% RSLogix 500 project CHIZOM SCADA MAIN.RSS %
PROJECT "UNTITLED"    % processor: MicroLogix 1000 %

PROGRAM FILES
  LAD 2 "MAIN_PROG"  36 rungs
  LAD 3 "USER_FAULT"  1 rungs
  LAD 4 "HSC_INT"  1 rungs
  LAD 5 "STI_INT"  1 rungs
  LAD 6, 7, 8, 9, 10, 11, 12, 13, 14, 15, 16: only END

DATA FILES
  O0 OUTPUT  1 elements
  I1 INPUT  2 elements
  S2 STATUS  33 elements
  B3 BINARY  32 elements
  T4 TIMER  40 elements
  C5 COUNTER  32 elements
  R6 CONTROL  16 elements
  N7 INTEGER  105 elements

LADDER 2 "MAIN_PROG"
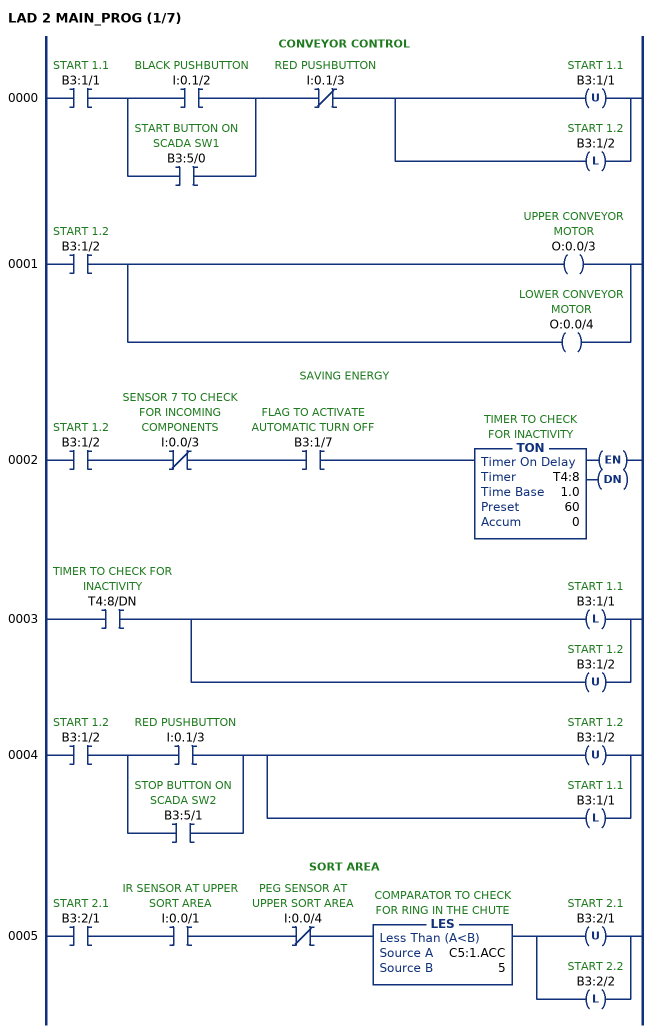
% Rung: 0 %
% TITLE: CONVEYOR CONTROL %
SOR XIC B3:1/1 BST XIC I:0.1/2 NXB XIC B3:5/0 BND XIO I:0.1/3 BST OTU B3:1/1 NXB OTL B3:1/2 BND EOR
%   B3:1/1  "START 1.1" %
%   I:0.1/2  "BLACK PUSHBUTTON" %
%   B3:5/0  SW1  "START BUTTON ON SCADA" %
%   I:0.1/3  "RED PUSHBUTTON" %
%   B3:1/2  "START 1.2" %
% Rung: 1 %
SOR XIC B3:1/2 BST OTE O:0.0/3 NXB OTE O:0.0/4 BND EOR
%   B3:1/2  "START 1.2" %
%   O:0.0/3  "UPPER CONVEYOR MOTOR" %
%   O:0.0/4  "LOWER CONVEYOR MOTOR" %
% Rung: 2 %
% SAVING ENERGY %
SOR XIC B3:1/2 XIO I:0.0/3 XIC B3:1/7 TON T4:8 1.0 60 0 EOR
%   B3:1/2  "START 1.2" %
%   I:0.0/3  "SENSOR 7 TO CHECK FOR INCOMING COMPONENTS" %
%   B3:1/7  "FLAG TO ACTIVATE AUTOMATIC TURN OFF" %
%   T4:8  "TIMER TO CHECK FOR INACTIVITY" %
% Rung: 3 %
SOR XIC T4:8/DN BST OTL B3:1/1 NXB OTU B3:1/2 BND EOR
%   T4:8  "TIMER TO CHECK FOR INACTIVITY" %
%   B3:1/1  "START 1.1" %
%   B3:1/2  "START 1.2" %
% Rung: 4 %
SOR XIC B3:1/2 BST XIC I:0.1/3 NXB XIC B3:5/1 BND BST OTU B3:1/2 NXB OTL B3:1/1 BND EOR
%   B3:1/2  "START 1.2" %
%   I:0.1/3  "RED PUSHBUTTON" %
%   B3:5/1  SW2  "STOP BUTTON ON SCADA" %
%   B3:1/1  "START 1.1" %
% Rung: 5 %
% TITLE: SORT AREA %
SOR XIC B3:2/1 XIC I:0.0/1 XIO I:0.0/4 LES C5:1.ACC 5 BST OTU B3:2/1 NXB OTL B3:2/2 BND EOR
%   B3:2/1  "START 2.1" %
%   I:0.0/1  "IR SENSOR AT UPPER SORT AREA" %
%   I:0.0/4  "PEG SENSOR AT UPPER SORT AREA" %
%   C5:1.ACC  "COMPARATOR TO CHECK FOR RING IN THE CHUTE" %
%   B3:2/2  "START 2.2" %

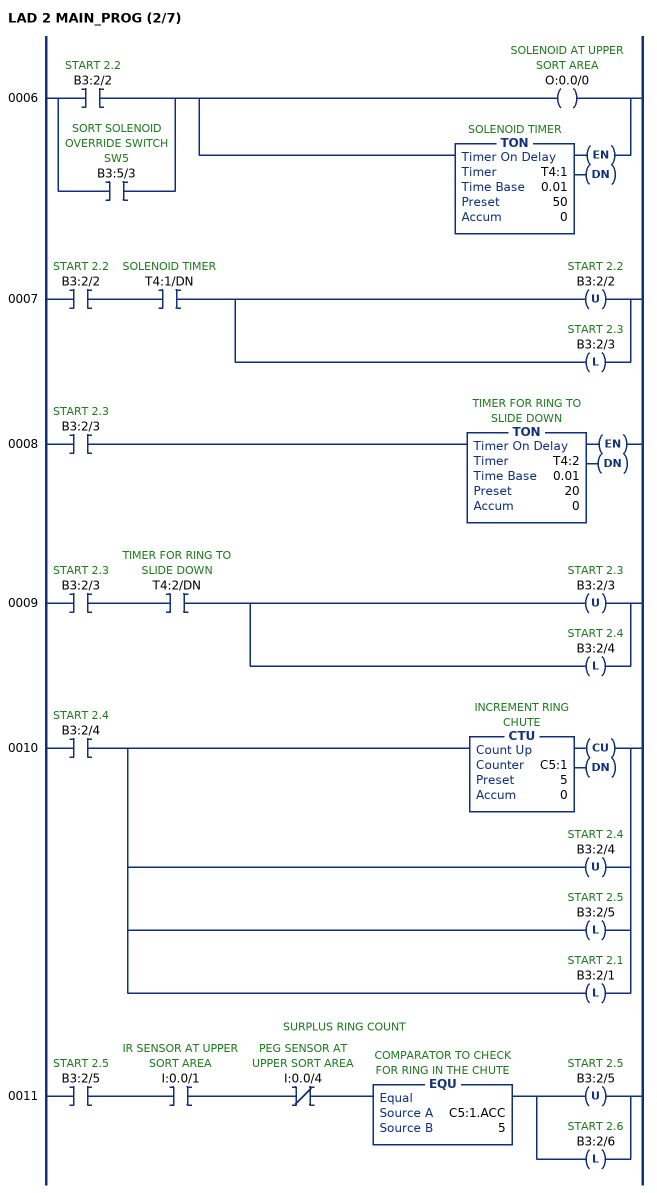
% Rung: 6 %
SOR BST XIC B3:2/2 NXB XIC B3:5/3 BND BST OTE O:0.0/0 NXB TON T4:1 0.01 50 0 BND EOR
%   B3:2/2  "START 2.2" %
%   B3:5/3  SW5  "SORT SOLENOID OVERRIDE SWITCH" %
%   O:0.0/0  "SOLENOID AT UPPER SORT AREA" %
%   T4:1  "SOLENOID TIMER" %
% Rung: 7 %
SOR XIC B3:2/2 XIC T4:1/DN BST OTU B3:2/2 NXB OTL B3:2/3 BND EOR
%   B3:2/2  "START 2.2" %
%   T4:1  "SOLENOID TIMER" %
%   B3:2/3  "START 2.3" %
% Rung: 8 %
SOR XIC B3:2/3 TON T4:2 0.01 20 0 EOR
%   B3:2/3  "START 2.3" %
%   T4:2  "TIMER FOR RING TO SLIDE DOWN" %
% Rung: 9 %
SOR XIC B3:2/3 XIC T4:2/DN BST OTU B3:2/3 NXB OTL B3:2/4 BND EOR
%   B3:2/3  "START 2.3" %
%   T4:2  "TIMER FOR RING TO SLIDE DOWN" %
%   B3:2/4  "START 2.4" %
% Rung: 10 %
SOR XIC B3:2/4 BST CTU C5:1 5 0 NXB BST OTU B3:2/4 NXB BST OTL B3:2/5 NXB OTL B3:2/1 BND BND BND EOR
%   B3:2/4  "START 2.4" %
%   C5:1  "INCREMENT RING CHUTE" %
%   B3:2/5  "START 2.5" %
%   B3:2/1  "START 2.1" %
% Rung: 11 %
% SURPLUS RING COUNT %
SOR XIC B3:2/5 XIC I:0.0/1 XIO I:0.0/4 EQU C5:1.ACC 5 BST OTU B3:2/5 NXB OTL B3:2/6 BND EOR
%   B3:2/5  "START 2.5" %
%   I:0.0/1  "IR SENSOR AT UPPER SORT AREA" %
%   I:0.0/4  "PEG SENSOR AT UPPER SORT AREA" %
%   C5:1.ACC  "COMPARATOR TO CHECK FOR RING IN THE CHUTE" %
%   B3:2/6  "START 2.6" %

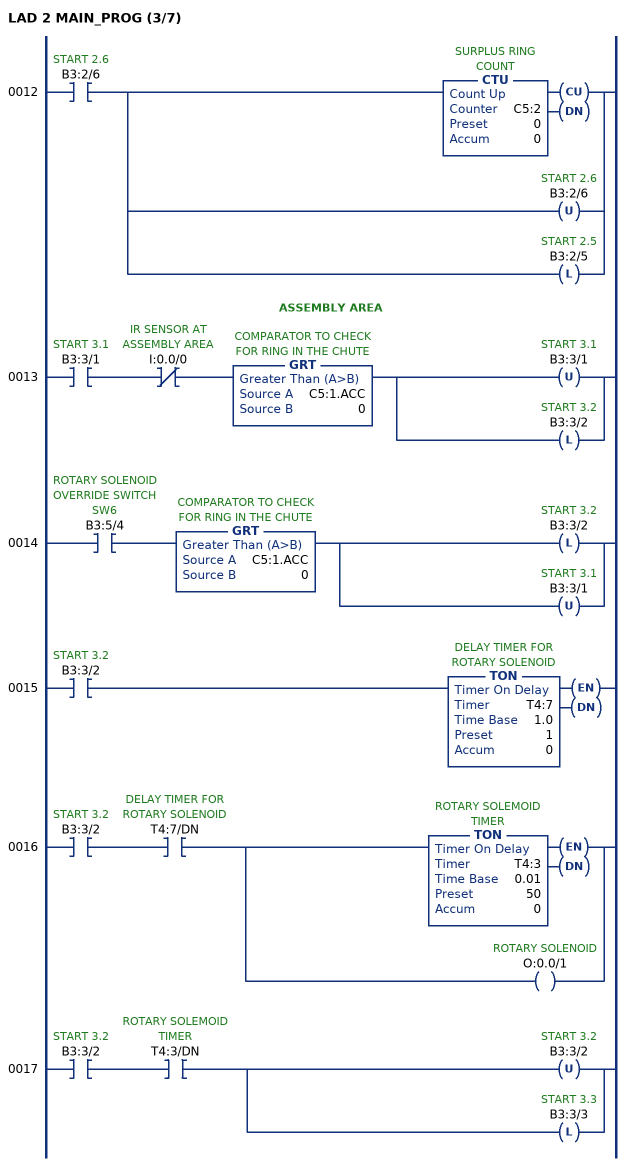
% Rung: 12 %
SOR XIC B3:2/6 BST CTU C5:2 0 0 NXB BST OTU B3:2/6 NXB OTL B3:2/5 BND BND EOR
%   B3:2/6  "START 2.6" %
%   C5:2  "SURPLUS RING COUNT" %
%   B3:2/5  "START 2.5" %
% Rung: 13 %
% TITLE: ASSEMBLY AREA %
SOR XIC B3:3/1 XIO I:0.0/0 GRT C5:1.ACC 0 BST OTU B3:3/1 NXB OTL B3:3/2 BND EOR
%   B3:3/1  "START 3.1" %
%   I:0.0/0  "IR SENSOR AT ASSEMBLY AREA" %
%   C5:1.ACC  "COMPARATOR TO CHECK FOR RING IN THE CHUTE" %
%   B3:3/2  "START 3.2" %
% Rung: 14 %
SOR XIC B3:5/4 GRT C5:1.ACC 0 BST OTL B3:3/2 NXB OTU B3:3/1 BND EOR
%   B3:5/4  SW6  "ROTARY SOLENOID OVERRIDE SWITCH" %
%   C5:1.ACC  "COMPARATOR TO CHECK FOR RING IN THE CHUTE" %
%   B3:3/2  "START 3.2" %
%   B3:3/1  "START 3.1" %
% Rung: 15 %
SOR XIC B3:3/2 TON T4:7 1.0 1 0 EOR
%   B3:3/2  "START 3.2" %
%   T4:7  "DELAY TIMER FOR ROTARY SOLENOID" %
% Rung: 16 %
SOR XIC B3:3/2 XIC T4:7/DN BST TON T4:3 0.01 50 0 NXB OTE O:0.0/1 BND EOR
%   B3:3/2  "START 3.2" %
%   T4:7  "DELAY TIMER FOR ROTARY SOLENOID" %
%   T4:3  "ROTARY SOLEMOID TIMER" %
%   O:0.0/1  "ROTARY SOLENOID" %
% Rung: 17 %
SOR XIC B3:3/2 XIC T4:3/DN BST OTU B3:3/2 NXB OTL B3:3/3 BND EOR
%   B3:3/2  "START 3.2" %
%   T4:3  "ROTARY SOLEMOID TIMER" %
%   B3:3/3  "START 3.3" %

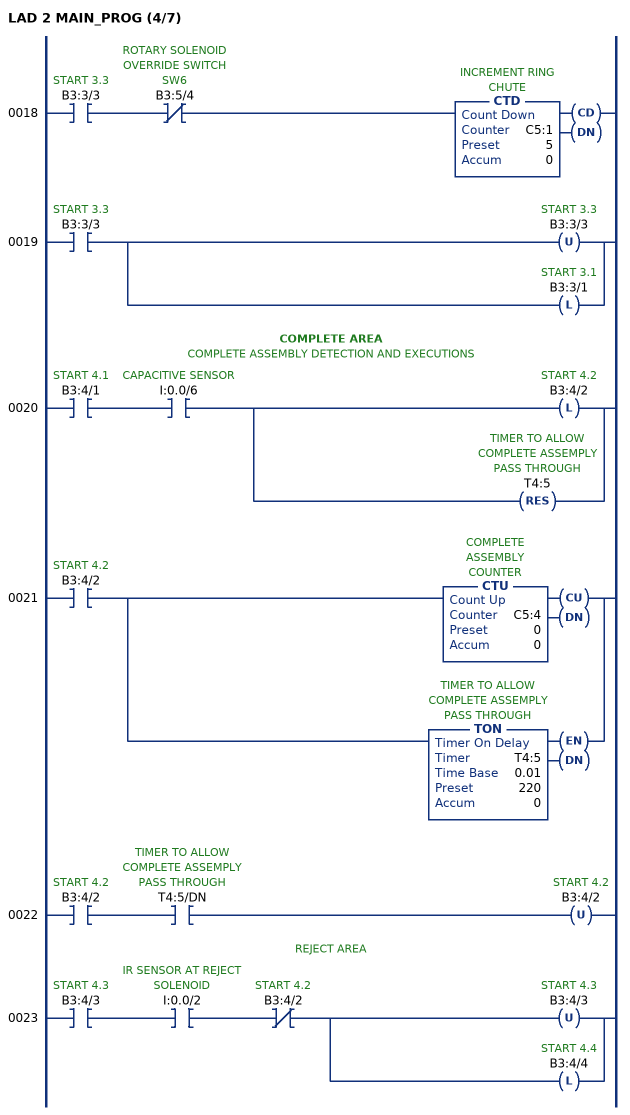
% Rung: 18 %
SOR XIC B3:3/3 XIO B3:5/4 CTD C5:1 5 0 EOR
%   B3:3/3  "START 3.3" %
%   B3:5/4  SW6  "ROTARY SOLENOID OVERRIDE SWITCH" %
%   C5:1  "INCREMENT RING CHUTE" %
% Rung: 19 %
SOR XIC B3:3/3 BST OTU B3:3/3 NXB OTL B3:3/1 BND EOR
%   B3:3/3  "START 3.3" %
%   B3:3/1  "START 3.1" %
% Rung: 20 %
% TITLE: COMPLETE AREA %
% COMPLETE ASSEMBLY DETECTION AND EXECUTIONS %
SOR XIC B3:4/1 XIC I:0.0/6 BST OTL B3:4/2 NXB RES T4:5 BND EOR
%   B3:4/1  "START 4.1" %
%   I:0.0/6  "CAPACITIVE SENSOR" %
%   B3:4/2  "START 4.2" %
%   T4:5  "TIMER TO ALLOW COMPLETE ASSEMPLY PASS THROUGH" %
% Rung: 21 %
SOR XIC B3:4/2 BST CTU C5:4 0 0 NXB TON T4:5 0.01 220 0 BND EOR
%   B3:4/2  "START 4.2" %
%   C5:4  "COMPLETE ASSEMBLY COUNTER" %
%   T4:5  "TIMER TO ALLOW COMPLETE ASSEMPLY PASS THROUGH" %
% Rung: 22 %
SOR XIC B3:4/2 XIC T4:5/DN OTU B3:4/2 EOR
%   B3:4/2  "START 4.2" %
%   T4:5  "TIMER TO ALLOW COMPLETE ASSEMPLY PASS THROUGH" %
% Rung: 23 %
% REJECT AREA %
SOR XIC B3:4/3 XIC I:0.0/2 XIO B3:4/2 BST OTU B3:4/3 NXB OTL B3:4/4 BND EOR
%   B3:4/3  "START 4.3" %
%   I:0.0/2  "IR SENSOR AT REJECT SOLENOID" %
%   B3:4/2  "START 4.2" %
%   B3:4/4  "START 4.4" %

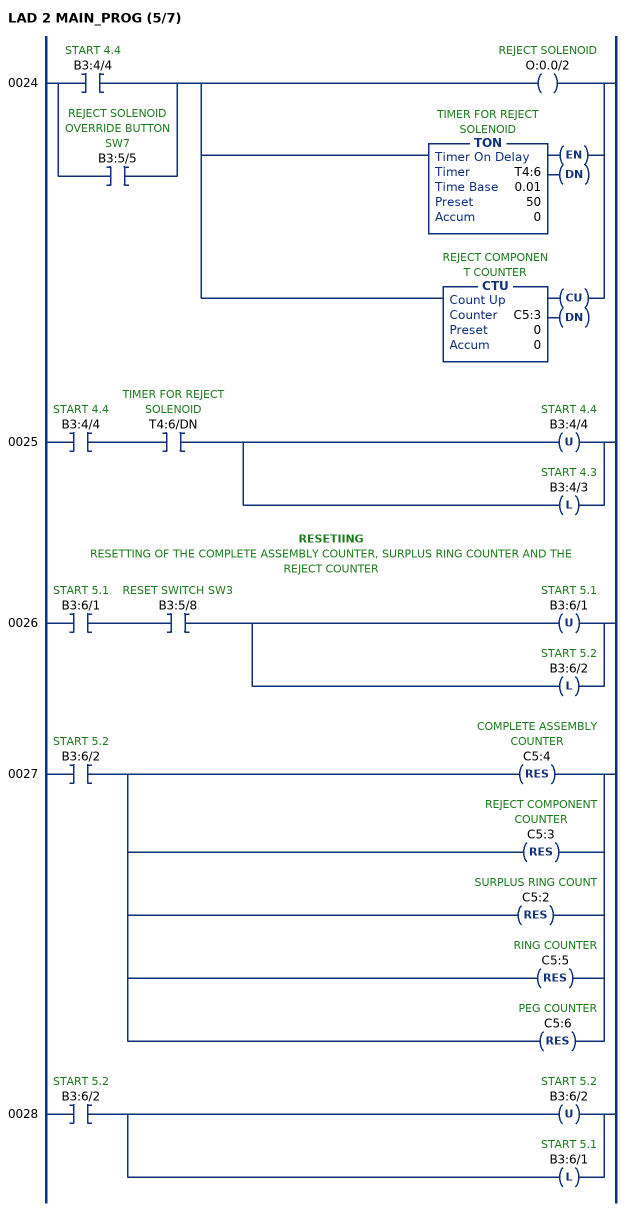
% Rung: 24 %
SOR BST XIC B3:4/4 NXB XIC B3:5/5 BND BST OTE O:0.0/2 NXB BST TON T4:6 0.01 50 0 NXB CTU C5:3 0 0 BND BND EOR
%   B3:4/4  "START 4.4" %
%   B3:5/5  SW7  "REJECT SOLENOID OVERRIDE BUTTON" %
%   O:0.0/2  "REJECT SOLENOID" %
%   T4:6  "TIMER FOR REJECT SOLENOID" %
%   C5:3  "REJECT COMPONENT COUNTER" %
% Rung: 25 %
SOR XIC B3:4/4 XIC T4:6/DN BST OTU B3:4/4 NXB OTL B3:4/3 BND EOR
%   B3:4/4  "START 4.4" %
%   T4:6  "TIMER FOR REJECT SOLENOID" %
%   B3:4/3  "START 4.3" %
% Rung: 26 %
% TITLE: RESETIING %
% RESETTING OF THE COMPLETE ASSEMBLY COUNTER, SURPLUS RING COUNTER AND THE REJECT COUNTER %
SOR XIC B3:6/1 XIC B3:5/8 BST OTU B3:6/1 NXB OTL B3:6/2 BND EOR
%   B3:6/1  "START 5.1" %
%   B3:5/8  SW3  "RESET SWITCH" %
%   B3:6/2  "START 5.2" %
% Rung: 27 %
SOR XIC B3:6/2 BST RES C5:4 NXB BST RES C5:3 NXB BST RES C5:2 NXB BST RES C5:5 NXB RES C5:6 BND BND BND BND EOR
%   B3:6/2  "START 5.2" %
%   C5:4  "COMPLETE ASSEMBLY COUNTER" %
%   C5:3  "REJECT COMPONENT COUNTER" %
%   C5:2  "SURPLUS RING COUNT" %
%   C5:5  "RING COUNTER" %
%   C5:6  "PEG COUNTER" %
% Rung: 28 %
SOR XIC B3:6/2 BST OTU B3:6/2 NXB OTL B3:6/1 BND EOR
%   B3:6/2  "START 5.2" %
%   B3:6/1  "START 5.1" %

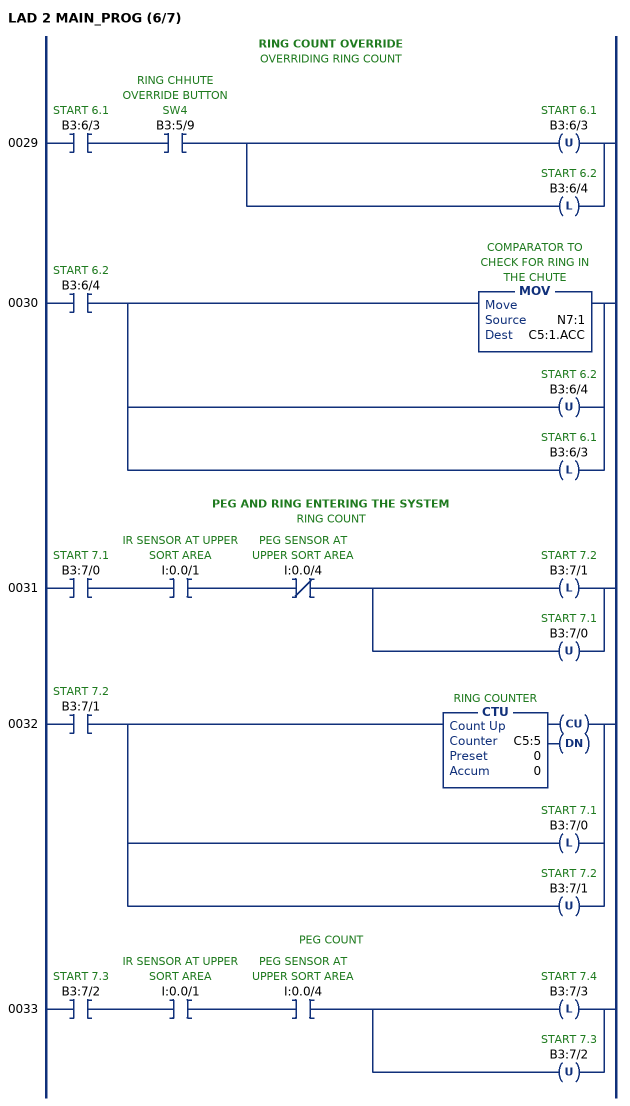
% Rung: 29 %
% TITLE: RING COUNT OVERRIDE %
% OVERRIDING RING COUNT %
SOR XIC B3:6/3 XIC B3:5/9 BST OTU B3:6/3 NXB OTL B3:6/4 BND EOR
%   B3:6/3  "START 6.1" %
%   B3:5/9  SW4  "RING CHHUTE OVERRIDE BUTTON" %
%   B3:6/4  "START 6.2" %
% Rung: 30 %
SOR XIC B3:6/4 BST MOV N7:1 C5:1.ACC NXB BST OTU B3:6/4 NXB OTL B3:6/3 BND BND EOR
%   B3:6/4  "START 6.2" %
%   N7:1  "DATA FROM SCADA SYSTEM" %
%   C5:1.ACC  "COMPARATOR TO CHECK FOR RING IN THE CHUTE" %
%   B3:6/3  "START 6.1" %
% Rung: 31 %
% TITLE: PEG AND RING ENTERING THE SYSTEM %
% RING COUNT %
SOR XIC B3:7/0 XIC I:0.0/1 XIO I:0.0/4 BST OTL B3:7/1 NXB OTU B3:7/0 BND EOR
%   B3:7/0  "START 7.1" %
%   I:0.0/1  "IR SENSOR AT UPPER SORT AREA" %
%   I:0.0/4  "PEG SENSOR AT UPPER SORT AREA" %
%   B3:7/1  "START 7.2" %
% Rung: 32 %
SOR XIC B3:7/1 BST CTU C5:5 0 0 NXB BST OTL B3:7/0 NXB OTU B3:7/1 BND BND EOR
%   B3:7/1  "START 7.2" %
%   C5:5  "RING COUNTER" %
%   B3:7/0  "START 7.1" %
% Rung: 33 %
% PEG COUNT %
SOR XIC B3:7/2 XIC I:0.0/1 XIC I:0.0/4 BST OTL B3:7/3 NXB OTU B3:7/2 BND EOR
%   B3:7/2  "START 7.3" %
%   I:0.0/1  "IR SENSOR AT UPPER SORT AREA" %
%   I:0.0/4  "PEG SENSOR AT UPPER SORT AREA" %
%   B3:7/3  "START 7.4" %

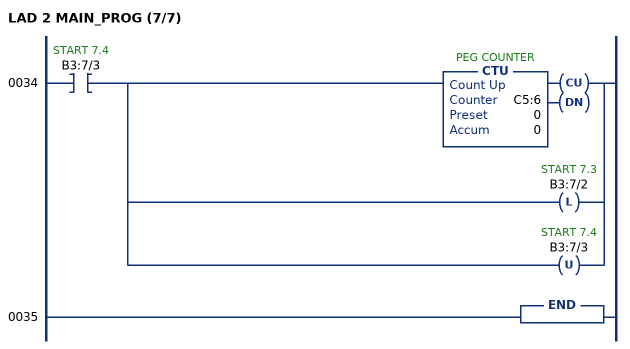
% Rung: 34 %
SOR XIC B3:7/3 BST CTU C5:6 0 0 NXB BST OTL B3:7/2 NXB OTU B3:7/3 BND BND EOR
%   B3:7/3  "START 7.4" %
%   C5:6  "PEG COUNTER" %
%   B3:7/2  "START 7.3" %
% Rung: 35 %
SOR END EOR

OTHER DOCUMENTED ADDRESSES
  B3:5/2  LED1

COMMENTS NOT ATTACHED TO A CURRENT RUNG
  C5:4: COMPLETE ASSEMBLY COUNTING
  C5:1.ACC: RING COUNT RESETING

DATA TABLE (non-zero values as saved)
DATA B3
% B3:0 % 0X0000 0X0002 0X0022 0X0002 0X000A 0X0000 0X000B 0X0005 0X0000 0X0000
DATA T4
% .PRE .ACC %
% T4:1 % 50 0
% T4:2 % 20 0
% T4:3 % 50 0
% T4:4 % 50 0
% T4:5 % 220 0
% T4:6 % 50 0
% T4:7 % 1 0
% T4:8 % 60 0
% T4:9 % 3 0
DATA C5
% .PRE .ACC %
% C5:1 % 5 0
